Staubli VAL3: new.pgx

public program new(string x_sName (dimensions=1), num& x_nResult[] (dimensions=1))
  local string l_sPrefix
  local num l_nResult
begin
  // new one
  if insert(pt:tTraj[x_sName])
    call pt:link_it(x_sName)
    pt:tTraj[x_sName].nIndexTool=saveData:nIndexTool
    x_nResult=0
    // set it
    bToSave=true
  else
    x_nResult=-1
  endIf
end
